TEXTLIST PDU_Surge_Status
  0 = 'HEALTHY'
  1 = 'ALARM'
   = ''
END_TEXTLIST

(* stored: Version 1.1.0.1, ProductVersion 3.1.4024.12
   TextList PDU_Surge_Status: Id {2a653566-2b9e-4684-a1ec-eca0fa218d32} *)
